Staubli VAL3: IoWriteRequest.pjx

--- IoWriteRequest.pjx ---
Parameters version=s7.7.2 stackSize=5000 millimeterUnit=true
Program file=start.pgx
Program file=stop.pgx
Data file=IoWriteRequest.dtx

--- IoWriteRequest.dtx ---
public num nCount
public num nType
public num nIndex
public num nValue
